VAR_GLOBAL
	bSafetyRun AT %Q*		:	BOOL;
	bSafetyErrorAck AT %Q*	:	BOOL;
	bSafetyComErr AT %I*	:	BOOL;
	bSafetyFbErr AT %I*		:	BOOL;
	bSafetyOutput AT %I*	:	BOOL;
END_VAR

(* stored: Version 1.1.0.1, ProductVersion 3.1.4024.6
   GVL GVL: Id {7bebd6dc-ffb7-477e-ab80-f99eaa86bb37} *)
